PROGRAM MAIN
VAR
END_VAR

END_PROGRAM

(* stored: Version 1.1.0.1
   POU MAIN: Id {58f0b558-9b57-4304-8b06-3750e1ce8787} *)
